# B&R Automation Studio project git_study
Automation Studio 4.5.2.102; technology packages: mappView 5.2.3

## Configuration 5AP1120

CPU 5PC901.TS77-00, AutomationRuntime D4.52, Build 4.1.2, Vc V4.52.0

### Task classes (Cpu.sw)
```
Cyclic#4 (cycle 1000000 us, tolerance 1000000 us):
  Snake <- Snake.prg
VcDataObjects: Visu <- Visu.dob
```

### Hardware
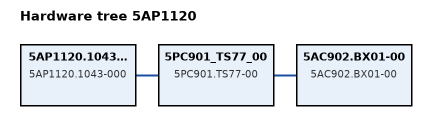
```
5AC902.BX01-00 : 5AC902.BX01-00 v1.1.1.0  [SY -> 5PC901_TS77_00.SY3]
5AP1120.1043-000 : 5AP1120.1043-000 v1.3.0.0
5PC901_TS77_00 : 5PC901.TS77-00 v2.0.0.0  [SY -> 5AP1120.1043-000.SY1]
  Connector IF1:
    AssignedOperatingSystem = ARemb
  Connector IF2:
    AssignedOperatingSystem = ARemb
  Connector IF3:
    AssignedOperatingSystem = ARemb
    ActivateDevice = 1
  Connector IF4:
    AssignedOperatingSystem = ARemb
    ActivateDevice = 1
  Connector IF5:
    AssignedOperatingSystem = ARemb
  Connector IF6:
    AssignedOperatingSystem = ARemb
  Connector IF7:
    AssignedOperatingSystem = ARemb
  Connector IF8:
    AssignedOperatingSystem = ARemb
  ConfigurationID = git_study_5AP1120
  Connector IF1:
    AssignedOperatingSystem = ARemb
  Connector IF2:
    AssignedOperatingSystem = ARemb
  Connector IF3:
    AssignedOperatingSystem = ARemb
    ActivateDevice = 1
  Connector IF4:
    AssignedOperatingSystem = ARemb
    ActivateDevice = 1
  Connector IF5:
    AssignedOperatingSystem = ARemb
  Connector IF6:
    AssignedOperatingSystem = ARemb
  Connector IF7:
    AssignedOperatingSystem = ARemb
  Connector IF8:
    AssignedOperatingSystem = ARemb
  ConfigurationID = git_study_5AP1120
  Cyclic4Duration = 1000000
  Cyclic4Tolerance = 1000000
  Simulation = 1
  ActivateOpcUa = 1
  OpcUaInformationModels_PV_Version = 1
```

## Configuration Config1

CPU 5PPC2100.BY01-000, AutomationRuntime D4.52, Build 4.1.2, Vc V4.52.0

### Task classes (Cpu.sw)
```

```

## Logical view

### Global.var - Global variables
```iecst
VAR
	Led : ARRAY[0..7] OF BOOL;
END_VAR
```

### Program Logical/Snake (ANSIC)

#### Cyclic.c
```c
#include <bur/plctypes.h>

#ifdef _DEFAULT_INCLUDES
	#include <AsDefault.h>
#endif

void _CYCLIC ProgramCyclic(void)
{

	Led[i] = 1;

	if ( i == 0 )
	{
		Led[7] = 0;
	}
	else
	{
		Led[i - 1] = 0;
	}
	i++;
	if (i > 7) i = 0;

}
```

- Visualisation Logical/mappView (not shown)

Listed in the project but not available here: Logical/Global.typ, Logical/Libraries
